// Write to HMI
//PGain:
IF NOT(G_Engineer_HMI.bPenable_dis_write) THEN
	G_Engineer_HMI.fProportionalgain_dis := fProportionalGain; // SKjønner ikke helt det her
ELSE
	fProportionalGain := G_Engineer_HMI.fProportionalgain_dis;
END_IF

//IGain: 
IF NOT(G_Engineer_HMI.bIenable_dis_write) THEN
	G_Engineer_HMI.fIntegralgain_dis := fIntegralGain;
ELSE
	fIntegralGain := G_Engineer_HMI.fIntegralgain_dis;
END_IF

fbPID_controller(
		ssMethodType := BOOL_TO_SINT(bEnable),
		error := fPosition_error,
		Int_error_threshold := G_PID_Tuning.Int_error_threshold,
		P_enable := G_Engineer_HMI.bPenable_dis,
		I_enable := G_Engineer_HMI.bIenable_dis,
		D_enable := FALSE,
		K_p := fProportionalGain,
		K_i := fIntegralGain,
		K_d := fDerivateGain,
		P_output => fProportinalGain_output,
		I_output => fIntegralGain_output,
		D_output => fDerivateGain_output
		);
		
			//Error times PGain
	fProportinalGain_output := fProportinalGain_output;
	G_PID_Tuning.fProportinalGain_output_dis := fProportinalGain_output;
	//Error times IGain
	fIntegralGain_output := fIntegralGain_output;
	G_PID_Tuning.fIntegralGain_output_dis := fIntegralGain_output;
	//Error times DGain
	fDerivateGain_output := fDerivateGain_output;
	G_PID_Tuning.fDerivateGain_output_dis := fDerivateGain_output;
	
	//Normalized Outputsignal
		
	fDisplacementControlSignal := LIMIT(-1, 1*(fProportinalGain_output + fIntegralGain_output + fDerivateGain_output), 1);
	G_PID_Tuning.PID_output_dis := fDisplacementControlSignal	;			
	
	IF ABS(fPosition_error) < 0.05 THEN
		bStartPosOK := TRUE;
	END_IF
		
ELSE
	bStartPosOK := FALSE;

END_IF

END_FUNCTION_BLOCK

// ---- PIDs/FB_PID_controller_old.TcPOU
FUNCTION_BLOCK FB_PID_controller_old
VAR_INPUT
	ssMethodType			: SINT;
	error					: LREAL;
	Int_error_threshold 	: LREAL;
	P_enable				: BOOL;
	I_enable				: BOOL;
	D_enable				: BOOL;
	K_p						: LREAL;
	K_i						: LREAL;
	K_d						: LREAL;
END_VAR
VAR_OUTPUT
	P_output: LREAL;
	I_output: LREAL;
	D_output: LREAL;
END_VAR
VAR
	rtb_TSamp: LREAL;
	c_DiscreteTimeIntegrator_DS: LREAL;
	UD_DSTATE: LREAL;
END_VAR



CASE ssMethodType OF
    0: 
        (* SystemInitialize for Atomic SubSystem: '<Root>/PID_controller' *)
        (* InitializeConditions for DiscreteIntegrator: '<S1>/Discrete-Time Integrator' *)
        c_DiscreteTimeIntegrator_DS := 0.0;
        (* InitializeConditions for UnitDelay: '<S2>/UD'
         *
         * Block description for '<S2>/UD':
         *  
         *  Store in Global RAM *)
        UD_DSTATE := 0.0;
        (* End of SystemInitialize for SubSystem: '<Root>/PID_controller' *)
    1: 
        (* Outputs for Atomic SubSystem: '<Root>/PID_controller' *)
        (* Switch: '<S1>/Switch' *)

        IF P_enable THEN 
            (* Outport: '<Root>/P_output' incorporates:
             *  Product: '<S1>/Product' *)
            P_output := LIMIT(-1, K_p * error, 1);
        ELSE 
            (* Outport: '<Root>/P_output' incorporates:
             *  Constant: '<S1>/Constant' *)
            P_output := 0.0;
        END_IF;

        (* End of Switch: '<S1>/Switch' *)
        

        (* Switch: '<S1>/Switch1' *)

        IF I_enable THEN 
            (* Outport: '<Root>/I_output' incorporates:
             *  DiscreteIntegrator: '<S1>/Discrete-Time Integrator' *)
            I_output := c_DiscreteTimeIntegrator_DS;
        ELSE 
            (* Outport: '<Root>/I_output' incorporates:
             *  Constant: '<S1>/Constant1' *)
            I_output := 0.0;
        END_IF;

        (* End of Switch: '<S1>/Switch1' *)
        

        (* SampleTimeMath: '<S2>/TSamp' incorporates:
         *  Product: '<S1>/Product2'
         *
         * About '<S2>/TSamp':
         *  y = u * K where K = 1 / ( w * Ts )
         *   *)
        rtb_TSamp := (K_d * error) * 100.0;
        (* Switch: '<S1>/Switch2' *)

        IF D_enable THEN 
            (* Outport: '<Root>/D_output' incorporates:
             *  Sum: '<S2>/Diff'
             *  UnitDelay: '<S2>/UD'
             *
             * Block description for '<S2>/Diff':
             *  
             *  Add in CPU
             *
             * Block description for '<S2>/UD':
             *  
             *  Store in Global RAM *)
            D_output := rtb_TSamp - UD_DSTATE;
        ELSE 
            (* Outport: '<Root>/D_output' incorporates:
             *  Constant: '<S1>/Constant2' *)
            D_output := 0.0;
        END_IF;

        (* End of Switch: '<S1>/Switch2' *)
        

        (* Update for DiscreteIntegrator: '<S1>/Discrete-Time Integrator' incorporates:
         *  Product: '<S1>/Product1' *)
       
		 //Anti windup med threshold verdi. Problem: Fører til oscillering
		(*IF ABS(error) < Int_error_threshold THEN
			c_DiscreteTimeIntegrator_DS := 0.0;
		ELSE
			c_DiscreteTimeIntegrator_DS := ((K_i * error) * 0.01) + c_DiscreteTimeIntegrator_DS;
		END_IF*)
		 c_DiscreteTimeIntegrator_DS := ((K_i * error) * 0.01) + c_DiscreteTimeIntegrator_DS;
		 
        (* Update for UnitDelay: '<S2>/UD'
         *
         * Block description for '<S2>/UD':
         *  
         *  Store in Global RAM *)
        UD_DSTATE := rtb_TSamp;
        (* End of Outputs for SubSystem: '<Root>/PID_controller' *)
END_CASE;

END_FUNCTION_BLOCK

// ---- Function Blocks/Currently not in use/FB_SecondaryControlSinus.TcPOU
FUNCTION_BLOCK FB_SecondaryControlSinus
VAR_INPUT
	ThetaRef 			: LREAL; // Kul
	fPosition 			: LREAL; 
	
END_VAR
VAR_OUTPUT
END_VAR
VAR
END_VAR

END_FUNCTION_BLOCK

// ---- PIDs/FB_PID_Controller_posref.TcPOU
FUNCTION_BLOCK FB_PID_Controller_posref
VAR_INPUT
	ssMethodType: SINT;
	fSignalReference: LREAL;
	fSignalFeedback: LREAL;
	fProportionalGain: LREAL;
	fIntegralGain: LREAL;
	bIntegralControlReset: BOOL;
	bActivateIntegralControl: BOOL;
	bEnable: BOOL;
	bActivateDerivativeControl: BOOL;
	fDerivativeGain: LREAL;
END_VAR
VAR_OUTPUT
	fClosedLoopSignal: LREAL;
	fSignalError: LREAL;
	P_out: LREAL;
	I_out: LREAL;
	D_out: LREAL;
END_VAR
VAR
	rtb_TSamp: LREAL;
	rtb_Sum5: LREAL;
	rtb_Saturation: LREAL;
	c_DiscreteTimeIntegrator1_D: LREAL;
	UD_DSTATE: LREAL;
END_VAR



CASE ssMethodType OF
    0: 
        (* SystemInitialize for Atomic SubSystem: '<Root>/FB_PID_new' *)
        (* InitializeConditions for DiscreteIntegrator: '<S1>/Discrete-Time Integrator1' *)
        c_DiscreteTimeIntegrator1_D := 0.0;
        (* InitializeConditions for UnitDelay: '<S2>/UD'
         *
         * Block description for '<S2>/UD':
         *  
         *  Store in Global RAM *)
        UD_DSTATE := 0.0;
        (* End of SystemInitialize for SubSystem: '<Root>/FB_PID_new' *)
    1: 
        (* Outputs for Atomic SubSystem: '<Root>/FB_PID_new' *)
        (* Sum: '<S1>/Sum' *)
        fSignalError := fSignalReference - fSignalFeedback;
        (* Product: '<S1>/Product' *)
        P_out := fProportionalGain * fSignalError;
        (* DiscreteIntegrator: '<S1>/Discrete-Time Integrator1' *)

        IF bIntegralControlReset THEN 
            c_DiscreteTimeIntegrator1_D := 0.0;
        END_IF;

        (* Switch: '<S1>/Switch2' incorporates:
         *  Constant: '<S1>/Constant'
         *  DiscreteIntegrator: '<S1>/Discrete-Time Integrator1' *)

        IF bActivateIntegralControl THEN 
            I_out := c_DiscreteTimeIntegrator1_D;
        ELSE 
            I_out := 0.0;
        END_IF;

        (* End of Switch: '<S1>/Switch2' *)
        

        (* SampleTimeMath: '<S2>/TSamp'
         *
         * About '<S2>/TSamp':
         *  y = u * K where K = 1 / ( w * Ts )
         *   *)
        rtb_TSamp := fDerivativeGain * 100.0;
        (* Switch: '<S1>/Switch3' incorporates:
         *  Constant: '<S1>/Constant2'
         *  Sum: '<S2>/Diff'
         *  UnitDelay: '<S2>/UD'
         *
         * Block description for '<S2>/Diff':
         *  
         *  Add in CPU
         *
         * Block description for '<S2>/UD':
         *  
         *  Store in Global RAM *)

        IF bActivateDerivativeControl THEN 
            D_out := rtb_TSamp - UD_DSTATE;
        ELSE 
            D_out := 0.0;
        END_IF;

        (* End of Switch: '<S1>/Switch3' *)
        

        (* Sum: '<S1>/Sum5' *)
        rtb_Sum5 := (P_out + I_out) + D_out;
        (* Saturate: '<S1>/Saturation' *)

        IF rtb_Sum5 > 1.0 THEN 
            rtb_Saturation := 1.0;
        ELSIF rtb_Sum5 >= -1.0 THEN 
            rtb_Saturation := rtb_Sum5;
        ELSE 
            rtb_Saturation := -1.0;
        END_IF;

        (* End of Saturate: '<S1>/Saturation' *)
        

        (* Switch: '<S1>/Switch1' *)

        IF bEnable THEN 
            (* Outport: '<Root>/fClosedLoopSignal' *)
            fClosedLoopSignal := rtb_Saturation;
        ELSE 
            (* Outport: '<Root>/fClosedLoopSignal' incorporates:
             *  Constant: '<S1>/Constant1' *)
            fClosedLoopSignal := 0.0;
        END_IF;

        (* End of Switch: '<S1>/Switch1' *)
        

        (* Update for DiscreteIntegrator: '<S1>/Discrete-Time Integrator1' incorporates:
         *  Product: '<S1>/Divide'
         *  Product: '<S1>/Product1'
         *  Sum: '<S1>/Sum1'
         *  Sum: '<S1>/Sum3' *)
        c_DiscreteTimeIntegrator1_D := (((((rtb_Saturation - rtb_Sum5) / fProportionalGain) + fSignalError) * fIntegralGain) * 0.01) + c_DiscreteTimeIntegrator1_D;

        IF c_DiscreteTimeIntegrator1_D > 1.0 THEN 
            c_DiscreteTimeIntegrator1_D := 1.0;
        ELSIF c_DiscreteTimeIntegrator1_D < -1.0 THEN 
            c_DiscreteTimeIntegrator1_D := -1.0;
        END_IF;

        (* End of Update for DiscreteIntegrator: '<S1>/Discrete-Time Integrator1' *)
        

        (* Update for UnitDelay: '<S2>/UD'
         *
         * Block description for '<S2>/UD':
         *  
         *  Store in Global RAM *)
        UD_DSTATE := rtb_TSamp;
        (* End of Outputs for SubSystem: '<Root>/FB_PID_new' *)
END_CASE;

END_FUNCTION_BLOCK

// ---- PIDs/FB_PID_SC.TcPOU
FUNCTION_BLOCK FB_PID_SC
VAR_INPUT
	ssMethodType: SINT;
	fSignalReference: LREAL;
	fSignalFeedback: LREAL;
	fProportionalGain: LREAL;
	fIntegralGain: LREAL;
	bIntegralControlReset: BOOL;
	bActivateIntegralControl: BOOL;
	bEnable: BOOL;
	bActivateDerivativeControl: BOOL;
	fDerivativeGain: LREAL;
END_VAR
VAR_OUTPUT
	fClosedLoopSignal: LREAL;
	fSignalError: LREAL;
	P_out: LREAL;
	I_out: LREAL;
	D_out: LREAL;
END_VAR
VAR
	rtb_TSamp: LREAL;
	rtb_Sum5: LREAL;
	rtb_Saturation: LREAL;
	c_DiscreteTimeIntegrator1_D: LREAL;
	UD_DSTATE: LREAL;
END_VAR



CASE ssMethodType OF
    0: 
        (* SystemInitialize for Atomic SubSystem: '<Root>/FB_PID_SC' *)
        (* InitializeConditions for DiscreteIntegrator: '<S1>/Discrete-Time Integrator1' *)
        c_DiscreteTimeIntegrator1_D := 0.0;
        (* InitializeConditions for UnitDelay: '<S2>/UD'
         *
         * Block description for '<S2>/UD':
         *  
         *  Store in Global RAM *)
        UD_DSTATE := 0.0;
        (* End of SystemInitialize for SubSystem: '<Root>/FB_PID_SC' *)
    1: 
        (* Outputs for Atomic SubSystem: '<Root>/FB_PID_SC' *)
        (* Sum: '<S1>/Sum' *)
        fSignalError := fSignalReference - fSignalFeedback;
        (* Product: '<S1>/Product' *)
        P_out := fProportionalGain * fSignalError;
        (* DiscreteIntegrator: '<S1>/Discrete-Time Integrator1' *)

        IF bIntegralControlReset THEN 
            c_DiscreteTimeIntegrator1_D := 0.0;
        END_IF;

        (* Switch: '<S1>/Switch2' incorporates:
         *  Constant: '<S1>/Constant'
         *  DiscreteIntegrator: '<S1>/Discrete-Time Integrator1' *)

        IF bActivateIntegralControl THEN 
            I_out := c_DiscreteTimeIntegrator1_D;
        ELSE 
            I_out := 0.0;
        END_IF;

        (* End of Switch: '<S1>/Switch2' *)
        

        (* SampleTimeMath: '<S2>/TSamp'
         *
         * About '<S2>/TSamp':
         *  y = u * K where K = 1 / ( w * Ts )
         *   *)
        rtb_TSamp := fDerivativeGain * 100.0;
        (* Switch: '<S1>/Switch3' incorporates:
         *  Constant: '<S1>/Constant2'
         *  Sum: '<S2>/Diff'
         *  UnitDelay: '<S2>/UD'
         *
         * Block description for '<S2>/Diff':
         *  
         *  Add in CPU
         *
         * Block description for '<S2>/UD':
         *  
         *  Store in Global RAM *)

        IF bActivateDerivativeControl THEN 
            D_out := rtb_TSamp - UD_DSTATE;
        ELSE 
            D_out := 0.0;
        END_IF;

        (* End of Switch: '<S1>/Switch3' *)
        

        (* Sum: '<S1>/Sum5' *)
        rtb_Sum5 := (P_out + I_out) + D_out;
        (* Saturate: '<S1>/Saturation' *)

        IF rtb_Sum5 > 1.0 THEN 
            rtb_Saturation := 1.0;
        ELSIF rtb_Sum5 >= -1.0 THEN 
            rtb_Saturation := rtb_Sum5;
        ELSE 
            rtb_Saturation := -1.0;
        END_IF;

        (* End of Saturate: '<S1>/Saturation' *)
        

        (* Switch: '<S1>/Switch1' *)

        IF bEnable THEN 
            (* Outport: '<Root>/fClosedLoopSignal' *)
            fClosedLoopSignal := rtb_Saturation;
        ELSE 
            (* Outport: '<Root>/fClosedLoopSignal' incorporates:
             *  Constant: '<S1>/Constant1' *)
            fClosedLoopSignal := 0.0;
        END_IF;

        (* End of Switch: '<S1>/Switch1' *)
        

        (* Update for DiscreteIntegrator: '<S1>/Discrete-Time Integrator1' incorporates:
         *  Product: '<S1>/Divide'
         *  Product: '<S1>/Product1'
         *  Sum: '<S1>/Sum1'
         *  Sum: '<S1>/Sum3' *)
        c_DiscreteTimeIntegrator1_D := (((((rtb_Saturation - rtb_Sum5) / fProportionalGain) + fSignalError) * fIntegralGain) * 0.01) + c_DiscreteTimeIntegrator1_D;

        IF c_DiscreteTimeIntegrator1_D > 1.0 THEN 
            c_DiscreteTimeIntegrator1_D := 1.0;
        ELSIF c_DiscreteTimeIntegrator1_D < -1.0 THEN 
            c_DiscreteTimeIntegrator1_D := -1.0;
        END_IF;

        (* End of Update for DiscreteIntegrator: '<S1>/Discrete-Time Integrator1' *)
        

        (* Update for UnitDelay: '<S2>/UD'
         *
         * Block description for '<S2>/UD':
         *  
         *  Store in Global RAM *)
        UD_DSTATE := rtb_TSamp;
        (* End of Outputs for SubSystem: '<Root>/FB_PID_SC' *)
END_CASE;

END_FUNCTION_BLOCK

// ---- Engineer_HMI.TcVIS
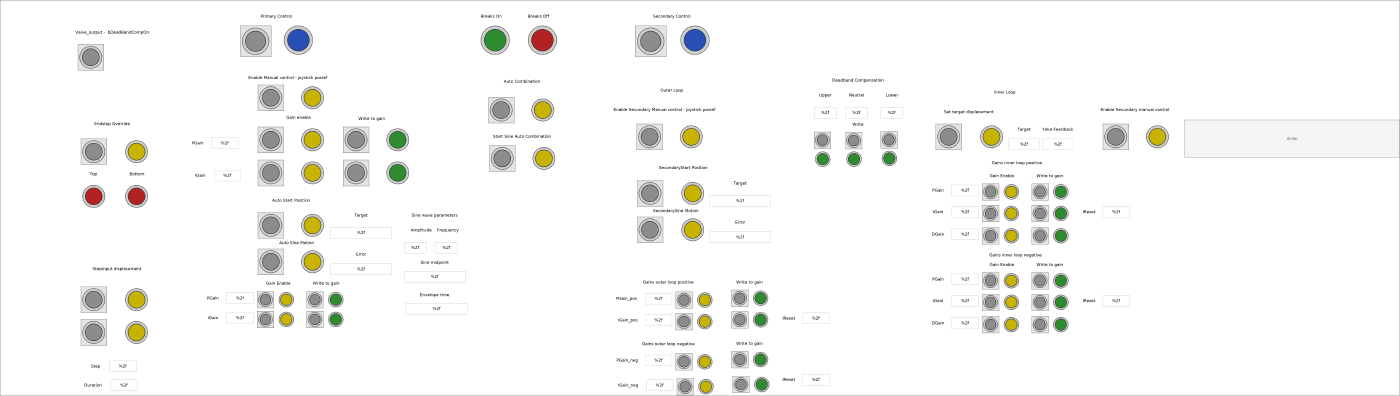
VISUALIZATION Engineer_HMI  // 3763x1065
    PushSwitch (209,119 70x70), variable: G_Parameters.stParam.bWinchDeadBandCompOn, behaviour: TOGGLE, style: Switch-PushSwitch-Gray
    Label (169,72 265x30), "Valve_output - bDeadBandCompOn"
    PushSwitch (217,373 70x70), variable: G_Engineer_HMI.bEndStopOverride, behaviour: TOGGLE, style: Switch-PushSwitch-Gray
    Lamp1 (332,373 70x70), variable: G_Engineer_HMI.bEndStopOverride, style: Lamp-Lamp1-Yellow
    Label (169,318 265x30), "Endstop Override"
    Lamp1 (217,493 70x70), variable: G_Engineer_HMI.bEndStopUpActive, style: Lamp-Lamp1-Red
    Label (217,453 68x30), "Top"
    Label (334,453 68x30), "Bottom"
    Lamp1 (332,493 70x70), variable: G_Engineer_HMI.bEndStopDownActive, style: Lamp-Lamp1-Red
    PushSwitch (217,771 70x70), variable: G_Engineer_HMI.bStepInput, behaviour: TOGGLE, style: Switch-PushSwitch-Gray
    Lamp1 (332,771 70x70), variable: G_Engineer_HMI.bStepInput, style: Lamp-Lamp1-Yellow
    Label (182,708 265x30), "StepInput displacement"
    Label (236,970 43x30), "Step"
    Textfield (294,970 72x30), "%2f", text variable: G_Engineer_HMI.fStepInput
        OnMouseClick: write G_Engineer_HMI.fStepInput via Default
    Label (219,1021 63x30), "Duration"
    Textfield (297,1021 72x30), "%2f", text variable: G_Engineer_HMI.fDuration
        OnMouseClick: write G_Engineer_HMI.fDuration via Default
    PushSwitch (217,859 70x70), variable: G_Engineer_HMI.bStartStepInput, behaviour: TOGGLE, style: Switch-PushSwitch-Gray
    Lamp1 (332,859 70x70), variable: G_Engineer_HMI.bStartStepInput, style: Lamp-Lamp1-Yellow
    Lamp1 (751,63 102x90), variable: G_Engineer_HMI.bPrimary_Control_active, style: Lamp-Lamp1-Blue
    PushSwitch (2515,333 70x70), variable: G_Engineer_HMI.bDisplacement_target_active, behaviour: TOGGLE, style: Switch-PushSwitch-Gray
    Lamp1 (2630,333 70x70), variable: G_Engineer_HMI.bDisplacement_target_active, style: Lamp-Lamp1-Yellow
    Label (2710,333 85x30), "Target"
    Label (2500,497 43x30), "PGain"
    Label (2500,286 209x30), "Set target displacement"
    Textfield (2710,373 85x30), "%2f", text variable: G_Engineer_HMI.fDisplacement_target
        OnMouseClick: write G_Engineer_HMI.fDisplacement_target via Default
    PushSwitch (2640,491 45x50), variable: G_Engineer_HMI.bPenable_IL, behaviour: TOGGLE, style: Switch-PushSwitch-Gray
    Lamp1 (2695,491 47x50), variable: G_Engineer_HMI.bPenable_IL, style: Lamp-Lamp1-Yellow
    Textfield (2558,497 72x30), "%2f", text variable: G_Engineer_HMI.fPGain_IL_Pos
        OnMouseClick: write G_Engineer_HMI.fPGain_IL_Pos via Default
    Label (2773,458 98x30), "Write to gain"
    Label (2644,458 98x30), "Gain Enable"
    PushSwitch (2773,491 45x50), variable: G_Engineer_HMI.bPGain_IL_write_pos, behaviour: TOGGLE, style: Switch-PushSwitch-Gray
    Lamp1 (2828,491 47x50), variable: G_Engineer_HMI.bPGain_IL_write_pos, style: Lamp-Lamp1-Green
    Label (2500,555 43x30), "IGain"
    PushSwitch (2640,549 45x50), variable: G_Engineer_HMI.bIenable_IL, behaviour: TOGGLE, style: Switch-PushSwitch-Gray
    Lamp1 (2695,549 47x50), variable: G_Engineer_HMI.bIenable_IL, style: Lamp-Lamp1-Yellow
    Textfield (2558,555 72x30), "%2f", text variable: G_Engineer_HMI.fIGain_IL_Pos
        OnMouseClick: write G_Engineer_HMI.fIGain_IL_Pos via Default
    PushSwitch (2773,549 45x50), variable: G_Engineer_HMI.bIGain_IL_write_pos, behaviour: TOGGLE, style: Switch-PushSwitch-Gray
    Lamp1 (2828,549 47x50), variable: G_Engineer_HMI.bIGain_IL_write_pos, style: Lamp-Lamp1-Green
    Label (2500,615 43x30), "DGain"
    PushSwitch (2640,609 45x50), variable: G_Engineer_HMI.bDenable_IL, behaviour: TOGGLE, style: Switch-PushSwitch-Gray
    Lamp1 (2695,609 47x50), variable: G_Engineer_HMI.bDenable_IL, style: Lamp-Lamp1-Yellow
    Textfield (2558,615 72x30), "%2f", text variable: G_Engineer_HMI.fDGain_IL_Pos
        OnMouseClick: write G_Engineer_HMI.fDGain_IL_Pos via Default
    PushSwitch (2773,609 45x50), variable: G_Engineer_HMI.bDGain_IL_write_pos, behaviour: TOGGLE, style: Switch-PushSwitch-Gray
    Lamp1 (2828,609 47x50), variable: G_Engineer_HMI.bDGain_IL_write_pos, style: Lamp-Lamp1-Green
    PushSwitch (693,571 70x70), variable: G_Engineer_HMI.bAutoStartPosEnable, behaviour: TOGGLE, style: Switch-PushSwitch-Gray
    Lamp1 (805,571 70x70), variable: G_Engineer_HMI.bAutoStartPosEnable, style: Lamp-Lamp1-Yellow
    Label (678,524 209x30), "Auto Start Position"
    Textfield (888,611 165x30), "%2f", text variable: G_Engineer_HMI.fAutoStartPos_target
        OnMouseClick: write G_Engineer_HMI.fAutoStartPos_target via Default
    Label (551,787 43x30), "PGain"
    PushSwitch (691,781 45x50), variable: G_Engineer_HMI.bPenable_MOOG, behaviour: TOGGLE, style: Switch-PushSwitch-Gray
    Lamp1 (746,781 47x50), variable: G_Engineer_HMI.bPenable_MOOG, style: Lamp-Lamp1-Yellow
    Textfield (609,787 72x30), "%2f", text variable: G_Engineer_HMI.fPgain_MOOG
        OnMouseClick: write G_Engineer_HMI.fPgain_MOOG via Default
    PushSwitch (824,781 45x50), variable: G_Engineer_HMI.bPgain_MOOG_write, behaviour: TOGGLE, style: Switch-PushSwitch-Gray
    Lamp1 (879,781 47x50), variable: G_Engineer_HMI.bPgain_MOOG_write, style: Lamp-Lamp1-Green
    PushSwitch (693,669 70x70), variable: G_Engineer_HMI.bAutoSineMotionEnable, behaviour: TOGGLE, style: Switch-PushSwitch-Gray
    Lamp1 (805,669 70x70), variable: G_Engineer_HMI.bAutoSineMotionEnable, style: Lamp-Lamp1-Yellow
    Label (693,638 209x30), "Auto Sine Motion"
    Textfield (888,709 165x30), "%2f", text variable: G_Motion_Control.fPosition_error_SineMotion
    Label (551,840 43x30), "IGain"
    PushSwitch (691,834 45x50), variable: G_Engineer_HMI.bIenable_MOOG, behaviour: TOGGLE, style: Switch-PushSwitch-Gray
    Lamp1 (746,834 47x50), variable: G_Engineer_HMI.bIenable_MOOG, style: Lamp-Lamp1-Yellow
    Textfield (609,840 72x30), "%2f", text variable: G_Engineer_HMI.fIgain_MOOG
        OnMouseClick: write G_Engineer_HMI.fIgain_MOOG via Default
    PushSwitch (824,834 45x50), variable: G_Engineer_HMI.bIgain_MOOG_write, behaviour: TOGGLE, style: Switch-PushSwitch-Gray
    Lamp1 (879,834 47x50), variable: G_Engineer_HMI.bIgain_MOOG_write, style: Lamp-Lamp1-Green
    Label (888,564 165x30), "Target"
    Label (888,669 165x30), "Error"
    Label (1086,564 165x30), "Sine wave parameters"
    Textfield (1086,651 60x30), "%2f", text variable: G_Engineer_HMI.fAmp
        OnMouseClick: write G_Engineer_HMI.fAmp via Default
    Textfield (1170,651 60x30), "%2f", text variable: G_Engineer_HMI.fFreq
        OnMouseClick: write G_Engineer_HMI.fFreq via Default
    Label (1086,604 165x30), "Amplitude Frequency"
    Label (2801,333 85x30), "Yoke Feedback"
    Textfield (2801,373 85x30), "%2f", text variable: G_Sensors.fYokeNormalizedFeedback
    Textfield (1086,729 165x30), "%2f", text variable: G_Engineer_HMI.fSinemidpoint
        OnMouseClick: write G_Engineer_HMI.fSinemidpoint via Default
    Label (1086,691 165x30), "Sine midpoint"
    Label (828,747 98x30), "Write to gain"
    Label (699,747 98x30), "Gain Enable"
    PushSwitch (640,69 94x84), variable: G_Engineer_HMI.bPrimary_Control, behaviour: TAP, style: Switch-PushSwitch-Gray
    Label (638,29 209x30), "Primary Control"
    Lamp1 (1280,63 102x90), variable: NOT (G_IO.bOpenBrakes), style: Lamp-Lamp1-Green
    PushSwitch (1701,69 96x84), variable: G_Engineer_HMI.bSecondary_Control, behaviour: TAP, style: Switch-PushSwitch-Gray
    Label (1701,29 209x30), "Secondary Control"
    Label (1216,29 209x30), "Breaks On"
    Lamp1 (1817,63 102x90), variable: G_Engineer_HMI.bSecondary_Control_active, style: Lamp-Lamp1-Blue
    Lamp1 (1407,63 102x90), variable: G_IO.bOpenBrakes, style: Lamp-Lamp1-Red
    Label (1343,29 209x30), "Breaks Off"
    PushSwitch (2964,333 70x70), variable: G_Engineer_HMI.bJoystick_slider_active, behaviour: TOGGLE, style: Switch-PushSwitch-Gray
    Lamp1 (3076,333 70x70), variable: G_Engineer_HMI.bJoystick_slider_active, style: Lamp-Lamp1-Yellow
    Label (2930,280 241x30), "Enable Secundary manual control"
    PushSwitch (1712,485 70x70), variable: G_Engineer_HMI.bSecondaryStartPosEnable, behaviour: TOGGLE, style: Switch-PushSwitch-Gray
    Lamp1 (1827,485 70x70), variable: G_Engineer_HMI.bSecondaryStartPosEnable, style: Lamp-Lamp1-Yellow
    Label (1732,436 209x30), "SecondaryStart Position"
    Textfield (1907,525 165x30), "%2f", text variable: G_Engineer_HMI.fSecondaryStartPos_target
        OnMouseClick: write G_Engineer_HMI.fSecondaryStartPos_target via Default
    PushSwitch (1712,583 70x70), variable: G_Engineer_HMI.bSecondarySineMotionEnable, behaviour: TOGGLE, style: Switch-PushSwitch-Gray
    Lamp1 (1827,583 70x70), variable: G_Engineer_HMI.bSecondarySineMotionEnable, style: Lamp-Lamp1-Yellow
    Label (1712,552 209x30), "SecondarySine Motion"
    Textfield (1907,623 165x30), "%2f", text variable: G_Motion_Control.fPosition_error_StartDisplacement
    Label (1907,478 165x30), "Target"
    Label (1907,583 165x30), "Error"
    Label (510,370 43x30), "PGain"
    Textfield (568,370 72x30), "%2f", text variable: G_Engineer_HMI.fPGain_JoyPosref_PC
        OnMouseClick: write G_Engineer_HMI.fPGain_JoyPosref_PC via Default
    PushSwitch (693,228 70x70), variable: G_Engineer_HMI.bManualControl_enable, behaviour: TOGGLE, style: Switch-PushSwitch-Gray
    Lamp1 (805,228 70x70), variable: G_Engineer_HMI.bManualControl_enable, style: Lamp-Lamp1-Yellow
    Label (651,194 246x30), "Enable Manual control - joystick posref"
    Label (1086,778 165x30), "Envelope time"
    Textfield (1091,815 165x30), "%2f", text variable: G_Engineer_HMI.ft_ENV
        OnMouseClick: write G_Engineer_HMI.ft_ENV via Default
    PushSwitch (693,341 70x70), variable: G_Engineer_HMI.bPgain_enable_joy_posref, behaviour: TOGGLE, style: Switch-PushSwitch-Gray
    PushSwitch (693,430 70x70), variable: G_Engineer_HMI.bIgain_enable_joy_posref, behaviour: TOGGLE, style: Switch-PushSwitch-Gray
    Label (698,301 209x30), "Gain enable"
    Label (517,457 43x30), "IGain"
    Textfield (575,457 72x30), "%2f", text variable: G_Engineer_HMI.fIGain_JoyPosref_PC
        OnMouseClick: write G_Engineer_HMI.fIGain_JoyPosref_PC via Default
    Lamp1 (805,341 70x70), variable: G_Engineer_HMI.bPgain_enable_joy_posref, style: Lamp-Lamp1-Yellow
    Lamp1 (805,430 70x70), variable: G_Engineer_HMI.bIgain_enable_joy_posref, style: Lamp-Lamp1-Yellow
    PushSwitch (1711,333 70x70), variable: G_Engineer_HMI.bManual_Secondary_joyposref_enable, behaviour: TOGGLE, style: Switch-PushSwitch-Gray
    Lamp1 (1823,333 70x70), variable: G_Engineer_HMI.bManual_Secondary_joyposref_enable, style: Lamp-Lamp1-Yellow
    Label (1623,280 327x30), "Enable Secundary Manual control - joystick posref"
    Label (1633,744 327x30), "Gains outer loop positive"
    Label (1648,788 71x30), "PGain_pos"
    PushSwitch (1816,782 45x50), variable: G_Engineer_HMI.bPenable_OL, behaviour: TOGGLE, style: Switch-PushSwitch-Gray
    Lamp1 (1871,782 47x50), variable: G_Engineer_HMI.bPenable_OL, style: Lamp-Lamp1-Yellow
    Textfield (1734,788 72x30), "%2f", text variable: G_Engineer_HMI.fPGain_OL_Pos
        OnMouseClick: write G_Engineer_HMI.fPGain_OL_Pos via Default
    Label (1656,846 63x30), "IGain_pos"
    PushSwitch (1816,840 45x50), variable: G_Engineer_HMI.bIenable_OL, behaviour: TOGGLE, style: Switch-PushSwitch-Gray
    Lamp1 (1871,840 47x50), variable: G_Engineer_HMI.bIenable_OL, style: Lamp-Lamp1-Yellow
    Textfield (1734,846 72x30), "%2f", text variable: G_Engineer_HMI.fIGain_OL_Pos
        OnMouseClick: write G_Engineer_HMI.fIGain_OL_Pos via Default
    Label (2906,555 43x30), "IReset"
    Textfield (2964,555 72x30), "%2f", text variable: G_Engineer_HMI.fMaxerror_dis
        OnMouseClick: write G_Engineer_HMI.fMaxerror_dis via Default
    Label (895,304 209x30), "Write to gain"
    PushSwitch (922,341 70x70), variable: G_Engineer_HMI.bPgain_joy_posref_write, behaviour: TOGGLE, style: Switch-PushSwitch-Gray
    PushSwitch (922,430 70x70), variable: G_Engineer_HMI.bIgain_joy_posref_write, behaviour: TOGGLE, style: Switch-PushSwitch-Gray
    Lamp1 (1034,341 70x70), variable: G_Engineer_HMI.bPgain_joy_posref_write, style: Lamp-Lamp1-Green
    Lamp1 (1034,430 70x70), variable: G_Engineer_HMI.bIgain_joy_posref_write, style: Lamp-Lamp1-Green
    Label (1701,228 209x30), "Outer Loop"
    Label (2596,233 209x30), "Inner Loop"
    Label (1633,910 327x30), "Gains outer loop negative"
    Label (1653,954 66x30), "PGain_neg"
    PushSwitch (1816,948 45x50), variable: G_Engineer_HMI.bPenable_OL, behaviour: TOGGLE, style: Switch-PushSwitch-Gray
    Lamp1 (1871,948 47x50), variable: G_Engineer_HMI.bPenable_OL, style: Lamp-Lamp1-Yellow
    Textfield (1734,954 72x30), "%2f", text variable: G_Engineer_HMI.fPGain_OL_Neg
        OnMouseClick: write G_Engineer_HMI.fPGain_OL_Neg via Default
    Label (2500,736 43x30), "PGain"
    PushSwitch (2640,730 45x50), variable: G_Engineer_HMI.bPenable_IL, behaviour: TOGGLE, style: Switch-PushSwitch-Gray
    Lamp1 (2695,730 47x50), variable: G_Engineer_HMI.bPenable_IL, style: Lamp-Lamp1-Yellow
    Textfield (2558,736 72x30), "%2f", text variable: G_Engineer_HMI.fPGain_IL_Neg
        OnMouseClick: write G_Engineer_HMI.fPGain_IL_Neg via Default
    Label (2773,697 98x30), "Write to gain"
    Label (2644,697 98x30), "Gain Enable"
    PushSwitch (2773,730 45x50), variable: G_Engineer_HMI.bPGain_IL_write_neg, behaviour: TOGGLE, style: Switch-PushSwitch-Gray
    Lamp1 (2828,730 47x50), variable: G_Engineer_HMI.bPGain_IL_write_neg, style: Lamp-Lamp1-Green
    Label (2500,794 43x30), "IGain"
    PushSwitch (2640,788 45x50), variable: G_Engineer_HMI.bIenable_IL, behaviour: TOGGLE, style: Switch-PushSwitch-Gray
    Lamp1 (2695,788 47x50), variable: G_Engineer_HMI.bIenable_IL, style: Lamp-Lamp1-Yellow
    Textfield (2558,794 72x30), "%2f", text variable: G_Engineer_HMI.fIGain_IL_Neg
        OnMouseClick: write G_Engineer_HMI.fIGain_IL_Neg via Default
    PushSwitch (2773,788 45x50), variable: G_Engineer_HMI.bIGain_IL_write_neg, behaviour: TOGGLE, style: Switch-PushSwitch-Gray
    Lamp1 (2828,788 47x50), variable: G_Engineer_HMI.bIGain_IL_write_neg, style: Lamp-Lamp1-Green
    Label (2500,854 43x30), "DGain"
    PushSwitch (2640,848 45x50), variable: G_Engineer_HMI.bDenable_IL, behaviour: TOGGLE, style: Switch-PushSwitch-Gray
    Lamp1 (2695,848 47x50), variable: G_Engineer_HMI.bDenable_IL, style: Lamp-Lamp1-Yellow
    Textfield (2558,854 72x30), "%2f", text variable: G_Engineer_HMI.fDGain_IL_Neg
        OnMouseClick: write G_Engineer_HMI.fDGain_IL_Neg via Default
    PushSwitch (2773,848 45x50), variable: G_Engineer_HMI.bDGain_IL_write_neg, behaviour: TOGGLE, style: Switch-PushSwitch-Gray
    Lamp1 (2828,848 47x50), variable: G_Engineer_HMI.bDGain_IL_write_neg, style: Lamp-Lamp1-Green
    Label (2906,794 43x30), "IReset"
    Textfield (2964,794 72x30), "%2f", text variable: G_Engineer_HMI.fMaxerror_dis
        OnMouseClick: write G_Engineer_HMI.fMaxerror_dis via Default
    Label (2566,671 327x30), "Gains inner loop negative"
    Label (2570,423 327x30), "Gains inner loop positive"
    Label (1966,744 98x30), "Write to gain"
    PushSwitch (1966,777 45x50), variable: G_Engineer_HMI.bPGain_OL_write_pos, behaviour: TOGGLE, style: Switch-PushSwitch-Gray
    Lamp1 (2021,777 47x50), variable: G_Engineer_HMI.bPGain_OL_write_pos, style: Lamp-Lamp1-Green
    PushSwitch (1966,835 45x50), variable: G_Engineer_HMI.bIGain_OL_write_pos, behaviour: TOGGLE, style: Switch-PushSwitch-Gray
    Lamp1 (2021,835 47x50), variable: G_Engineer_HMI.bIGain_OL_write_pos, style: Lamp-Lamp1-Green
    Label (2099,841 43x30), "IReset"
    Textfield (2157,841 72x30), "%2f", text variable: G_Engineer_HMI.fMaxerror_dis
        OnMouseClick: write G_Engineer_HMI.fMaxerror_dis via Default
    Label (1966,909 98x30), "Write to gain"
    PushSwitch (1966,942 45x50), variable: G_Engineer_HMI.bPGain_OL_write_neg, behaviour: TOGGLE, style: Switch-PushSwitch-Gray
    Lamp1 (2021,942 47x50), variable: G_Engineer_HMI.bPGain_OL_write_neg, style: Lamp-Lamp1-Green
    Label (2099,1006 43x30), "IReset"
    Textfield (2157,1006 72x30), "%2f", text variable: G_Engineer_HMI.fMaxerror_dis
        OnMouseClick: write G_Engineer_HMI.fMaxerror_dis via Default
    Slider (3184,322 579x101), variable: G_Engineer_HMI.fDisplacement_target, scale 0..1
    Label (1656,1021 66x30), "IGain_neg"
    PushSwitch (1819,1015 45x50), variable: G_Engineer_HMI.bIenable_OL, behaviour: TOGGLE, style: Switch-PushSwitch-Gray
    Lamp1 (1874,1015 47x50), variable: G_Engineer_HMI.bIenable_OL, style: Lamp-Lamp1-Yellow
    Textfield (1737,1021 72x30), "%2f", text variable: G_Engineer_HMI.fIGain_OL_Neg
        OnMouseClick: write G_Engineer_HMI.fIGain_OL_Neg via Default
    PushSwitch (1969,1009 45x50), variable: G_Engineer_HMI.bIGain_OL_write_neg, behaviour: TOGGLE, style: Switch-PushSwitch-Gray
    Lamp1 (2024,1009 47x50), variable: G_Engineer_HMI.bIGain_OL_write_neg, style: Lamp-Lamp1-Green
    Textfield (2188,288 60x30), "%2f", text variable: G_Engineer_HMI.fUpperdeadband
        OnMouseClick: write G_Engineer_HMI.fUpperdeadband via Default
    Textfield (2272,288 60x30), "%2f", text variable: G_Engineer_HMI.fNeutraldeadband
        OnMouseClick: write G_Engineer_HMI.fNeutraldeadband via Default
    Label (2188,241 61x30), "Upper"
    Textfield (2367,288 60x30), "%2f", text variable: G_Engineer_HMI.fLowerdeadband
        OnMouseClick: write G_Engineer_HMI.fLowerdeadband via Default
    Label (2272,241 61x30), "Neutral"
    Label (2367,241 61x30), "Lower"
    Label (2202,201 209x30), "Deadband Compensation"
    Label (2257,320 98x30), "Write"
    PushSwitch (2188,352 45x50), variable: G_Engineer_HMI.bUpperWrite, behaviour: TOGGLE, style: Switch-PushSwitch-Gray
    Lamp1 (2188,403 47x50), variable: G_Engineer_HMI.bUpperWrite, style: Lamp-Lamp1-Green
    PushSwitch (2272,353 45x50), variable: G_Engineer_HMI.bNeutralWrite, behaviour: TOGGLE, style: Switch-PushSwitch-Gray
    Lamp1 (2272,403 47x50), variable: G_Engineer_HMI.bNeutralWrite, style: Lamp-Lamp1-Green
    PushSwitch (2367,351 45x50), variable: G_Engineer_HMI.bLowerWrite, behaviour: TOGGLE, style: Switch-PushSwitch-Gray
    Lamp1 (2367,401 47x50), variable: G_Engineer_HMI.bLowerWrite, style: Lamp-Lamp1-Green
    PushSwitch (1312,261 70x70), variable: G_Engineer_HMI.bCombinationActive, behaviour: TOGGLE, style: Switch-PushSwitch-Gray
    PushSwitch (1315,391 70x70), variable: G_Engineer_HMI.bAutoSineCombi, behaviour: TOGGLE, style: Switch-PushSwitch-Gray
    Lamp1 (1424,261 70x70), variable: G_Engineer_HMI.bCombinationActive, style: Lamp-Lamp1-Yellow
    Lamp1 (1427,391 70x70), variable: G_Engineer_HMI.bAutoSineCombi, style: Lamp-Lamp1-Yellow
    Label (1280,204 246x30), "Auto Combination"
    Label (1280,352 246x30), "Start Sine Auto Combination"
END_VISUALIZATION

// ---- GlobalTextList.TcGTLO
TEXTLIST GlobalTextList
  612 = ' Manual control - joystick posref - payload pos'
  736 = '%2f'
  336 = '%f'
  544 = '1'
  815 = '3'
  190 = 'Amplitude    Frequency'
  818 = 'Auto Combination'
  506 = 'Auto Sine Motion'
  877 = 'Auto Start Position'
  422 = 'Bottom'
  30 = 'Breaks Off'
  328 = 'Breaks On'
  394 = 'Breaks Open'
  340 = 'Deadband Compensation'
  335 = 'DGain'
  151 = 'Displacement mode'
  535 = 'Duration'
  106 = 'Enable Manual control'
  817 = 'Enable Manual control - joystick posref'
  520 = 'Enable Secundary manual control'
  88 = 'Enable Secundary Manual control'
  922 = 'Enable Secundary Manual control - joystick posref'
  616 = 'EndStop Override'
  49 = 'Endstop Override'
  829 = 'Envelope time'
  101 = 'Error'
  647 = 'Gain Enable'
  282 = 'Gain enable'
  542 = 'Gains inner loop negative'
  623 = 'Gains inner loop positive'
  415 = 'Gains outer loop negative'
  100 = 'Gains outer loop positive'
  112 = 'IGain'
  482 = 'IGain_neg'
  108 = 'IGain_pos'
  152 = 'Inner Loop'
  105 = 'IReset'
  39 = 'Joystick slider'
  582 = 'Lower'
  45 = 'Manual control - joystick pos ref'
  809 = 'Manual secundary'
  509 = 'Manuel control - joystick pos ref'
  681 = 'Neutral'
  561 = 'Open Breaks'
  569 = 'Outer Loop'
  928 = 'PGain'
  58 = 'PGain_neg'
  977 = 'PGain_pos'
  590 = 'PGaiPGain'
  17 = 'Primary Control'
  404 = 'Secondary Control'
  64 = 'SecondarySine Motion'
  944 = 'SecondaryStart Position'
  999 = 'Set displacement'
  560 = 'Set target displacement'
  222 = 'Set your displacement  bDeadBandCompOn'
  556 = 'Sine midpoint'
  467 = 'Sine motion displacement'
  421 = 'Sine wave parameters'
  191 = 'Start Sine Auto Combination'
  122 = 'Step'
  564 = 'StepInput displacement'
  899 = 'Target'
  967 = 'Top'
  446 = 'Upper'
  739 = 'Valve_output -  bDeadBandCompOn'
  820 = 'Wave parameters'
  929 = 'Write'
  499 = 'Write to gain'
  921 = 'Yoke Feedback'
END_TEXTLIST
